FUNCTION_BLOCK Counter (* Basic Function Block Type *)
  (* Standard: 61499-2 *)
  (* Version 0.3, 2009-09-15, JHC, Holobloc Inc, Changed transition priorities. *)
  (* Version 0.2, 2003-12-04, JHC, Rockwell Automation, Renamed for better indexing. *)
  (* Version 0.1, 2002-11-05, JHC, Rockwell Automation, Corrected missing ST element in Algorithm REQ. *)
  (* Version 0.0, 2000-05-30, JHC, Rockwell Automation *)
  PACKAGE fb.rt.DIAS;
  IMPORT fb.datatype.*;
  IMPORT fb.rt.*;
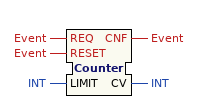
  EVENT_INPUT
    REQ; (* Normal Execution Request *)
    RESET;
  END_EVENT
  EVENT_OUTPUT
    CNF; (* Execution Confirmation *)
  END_EVENT
  VAR_INPUT
    LIMIT : INT;
  END_VAR
  VAR_OUTPUT
    CV : INT;
  END_VAR
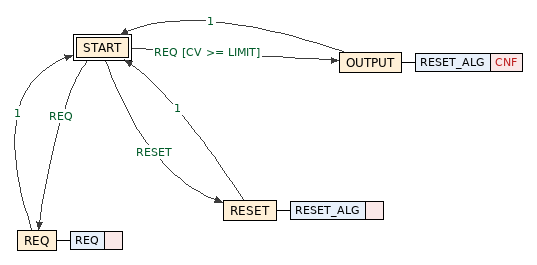
  EC_STATES
    START; (* Initial State *)
    REQ : REQ; (* Normal execution *)
    RESET : RESET_ALG;
    OUTPUT : RESET_ALG -> CNF;
  END_STATES
  EC_TRANSITIONS
    START TO REQ := REQ;
    REQ TO START := 1;
    START TO RESET := RESET;
    OUTPUT TO START := 1;
    START TO OUTPUT := REQ [CV >= LIMIT];
    RESET TO START := 1;
  END_TRANSITIONS
  ALGORITHM REQ IN ST:
CV := CV + 1;
  END_ALGORITHM
  ALGORITHM RESET_ALG IN ST:
CV := 0;
  END_ALGORITHM
END_FUNCTION_BLOCK
